ABB RobotStudio station: TFM_Robot.rspag

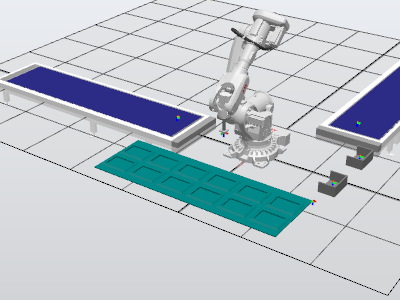
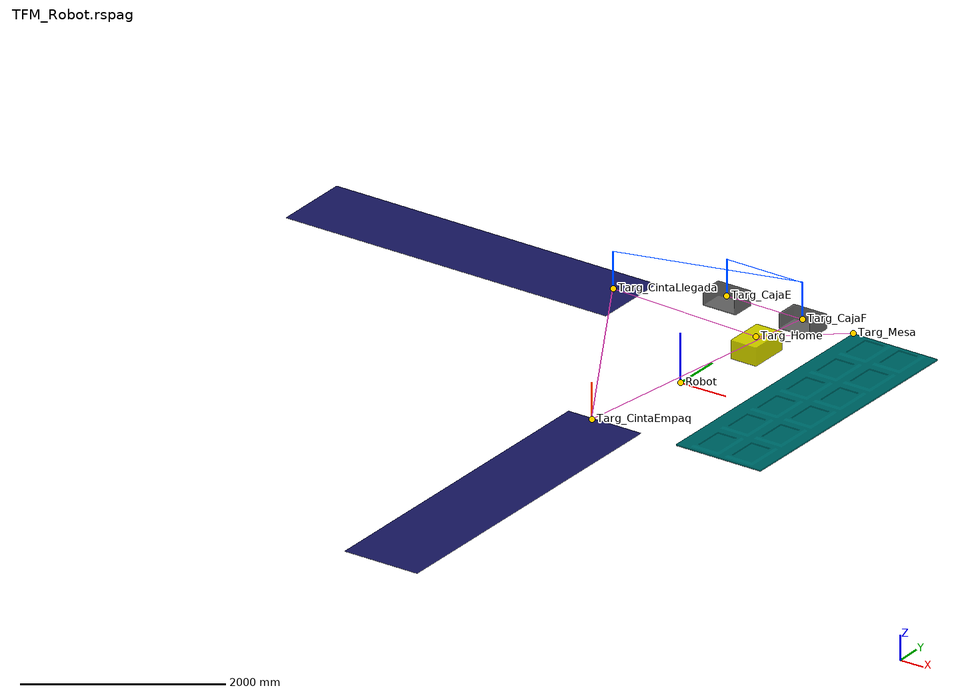
[picture v1: parts stored in the station drawn from their meshes, with robot base, taught points and paths (robot models come from the ABB library and are not in the file)]
--- station ---
Station TFM_Robot (saved by RobotStudio 24.2.10789.0)
Controller Controller_TFM
  mechanical unit ROB_1: Robot, 6 joints, base frame (0, 0, 0) mm
Layout (positions relative to the parent item):
  - Robot [mechanism] at (0, 0, 0) mm; joint values [0, -0.3937, 1.1224, 0, 0.8422, 1.5708] (rad or m)
      links: Base, Link1, Link2, Link3, Link4, Link5, Link6, LinkD1, LinkD2
  - GarraVentosas [mechanism] at (900, 0, 990) mm, rotated rx -180 ry 0 rz 90 deg
      TCP GarraVentosas at (0, 0, 240) mm
      links: GarraVentosas
  - MesaTrabajo [part] at (2000, 1500, 200) mm, rotated rx 90 ry 0 rz -90 deg, size 3000 x 35 x 1000 mm
  - CintaEmpaquetadora [part, from %ABB.RobotStudio.Models.Conveyors%\Conveyor 950 4000 h2.rslib] at (-455, -1200.38, -340.52) mm, rotated rx 0 ry 0 rz -90 deg
  - sup_CintaEmp [part] at (440.42, -1293.73, 94.49) mm, rotated rx 0 ry 0 rz 180 deg, size 864.5 x 3800 x 0 mm
  - sup_CintaGeneral [part] at (-1308.17, 600.35, 117.18) mm, rotated rx 0 ry 0 rz 90 deg, size 864.5 x 3800 x 0 mm
  - CintaGeneral [part, from %ABB.RobotStudio.Models.Conveyors%\Conveyor 950 4000 h2.rslib] at (-1231.46, 1484.09, -320.73) mm, rotated rx 0 ry 0 rz 180 deg
  - Surtidores_Cajas [part] at (205, 1630, 100) mm, rotated rx 90 ry 0 rz 0 deg, size 390 x 160 x 260 mm
  - Surtidores [part] at (-695, 1630, 100) mm, rotated rx 90 ry 0 rz 0 deg, size 390 x 160 x 260 mm
  - Ventosas [smart component] at (900, 0, 750) mm, rotated rx -180 ry 0 rz 90 deg
      signals: DI DI_Vacio, DI DI_Soplar, DO DO_Pieza, DI DI_VacioCaja, DI DI_SoplarCajas
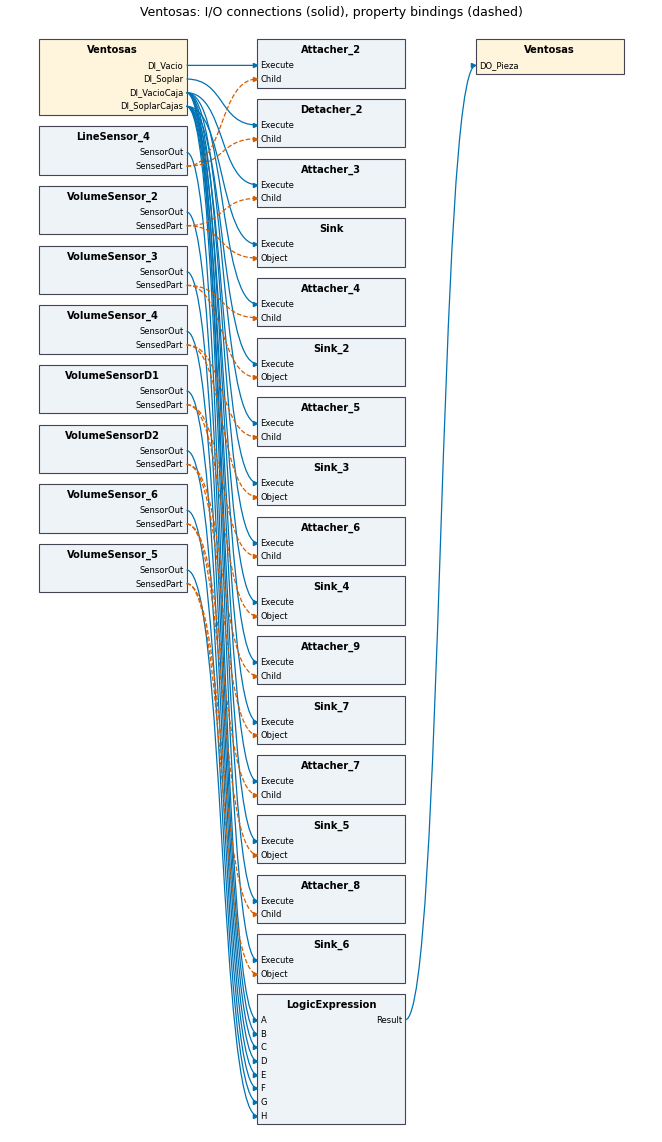
      connections:
        Ventosas.DI_Vacio -> Attacher_2.Execute
        Ventosas.DI_Soplar -> Detacher_2.Execute
        Ventosas.DI_VacioCaja -> Attacher_3.Execute
        Ventosas.DI_VacioCaja -> Attacher_4.Execute
        Ventosas.DI_VacioCaja -> Attacher_5.Execute
        Ventosas.DI_VacioCaja -> Attacher_6.Execute
        Ventosas.DI_VacioCaja -> Attacher_7.Execute
        Ventosas.DI_VacioCaja -> Attacher_8.Execute
        Ventosas.DI_SoplarCajas -> Sink.Execute
        Ventosas.DI_SoplarCajas -> Sink_2.Execute
        Ventosas.DI_SoplarCajas -> Sink_3.Execute
        Ventosas.DI_SoplarCajas -> Sink_4.Execute
        Ventosas.DI_SoplarCajas -> Sink_5.Execute
        Ventosas.DI_SoplarCajas -> Sink_6.Execute
        Ventosas.DI_VacioCaja -> Attacher_9.Execute
        Ventosas.DI_SoplarCajas -> Sink_7.Execute
        LineSensor_4.SensorOut -> LogicExpression.A
        VolumeSensor_2.SensorOut -> LogicExpression.B
        VolumeSensor_3.SensorOut -> LogicExpression.C
        VolumeSensor_4.SensorOut -> LogicExpression.D
        VolumeSensorD1.SensorOut -> LogicExpression.E
        VolumeSensorD2.SensorOut -> LogicExpression.F
        VolumeSensor_6.SensorOut -> LogicExpression.G
        VolumeSensor_5.SensorOut -> LogicExpression.H
        LogicExpression.Result -> Ventosas.DO_Pieza
        LineSensor_4.SensedPart => Attacher_2.Child
        LineSensor_4.SensedPart => Detacher_2.Child
        VolumeSensor_2.SensedPart => Attacher_3.Child
        VolumeSensor_2.SensedPart => Sink.Object
        VolumeSensor_3.SensedPart => Attacher_4.Child
        VolumeSensor_3.SensedPart => Sink_2.Object
        VolumeSensor_4.SensedPart => Attacher_5.Child
        VolumeSensor_4.SensedPart => Sink_3.Object
        VolumeSensorD1.SensedPart => Attacher_6.Child
        VolumeSensor_6.SensedPart => Attacher_7.Child
        VolumeSensor_5.SensedPart => Attacher_8.Child
        VolumeSensor_5.SensedPart => Sink_6.Object
        VolumeSensor_6.SensedPart => Sink_5.Object
        VolumeSensorD1.SensedPart => Sink_4.Object
        VolumeSensorD2.SensedPart => Attacher_9.Child
        VolumeSensorD2.SensedPart => Sink_7.Object
    - LineSensor_4 [smart component, from Components\LineSensor.rslib]
        properties: Start=[0.0199999999999999 0.02 -0.00999999999999998]; End=[0.0199999999999999 0.02 0.1]; Length=0.11; Radius=0.00476190476190476; Tag=(none); SensedPart=(none); SensedPoint=[0 0 0]
      - _sensorPart_ [part], size 9.5 x 9.5 x 110 mm
    - Attacher_2 [smart component, from Components\Attacher.rslib]
        properties: Parent=GarraVentosas; Flange=0; Child=(none); Mount=false; Offset=[0 0 0]; Orientation=[0 0 0]
    - Detacher_2 [smart component, from Components\Detacher.rslib]
        properties: Child=(none); KeepPosition=true
    - VolumeSensor_2 [smart component, from Components\VolumeSensor.rslib]
        properties: CornerPoint=[-0.220000006556705 -0.15000001063277 -0.00999992197537303]; Orientation=[0 0 0]; Length=0.44; Width=0.3; Height=0.2; Tag=PiezaA; PartialHit=true; SensedPart=(none)
      - _sensorPart_ [part], size 440 x 300 x 200 mm
    - VolumeSensor_3 [smart component, from Components\VolumeSensor.rslib] at (-100, 0, 0) mm
        properties: CornerPoint=[-0.120000006556705 -0.150000009019282 -0.00999992620903045]; Orientation=[0 0 0]; Length=0.44; Width=0.3; Height=0.2; Tag=PiezaB; PartialHit=true; SensedPart=(none)
      - _sensorPart_ [part], size 440 x 300 x 200 mm
    - VolumeSensor_4 [smart component, from Components\VolumeSensor.rslib] at (-200, 0, 0) mm
        properties: CornerPoint=[-0.0200000065567047 -0.150000007405794 -0.00999993044268799]; Orientation=[0 0 0]; Length=0.44; Width=0.3; Height=0.2; Tag=PiezaC; PartialHit=true; SensedPart=(none)
      - _sensorPart_ [part], size 440 x 300 x 200 mm
    - VolumeSensor_5 [smart component, from Components\VolumeSensor.rslib] at (-300, 0, 0) mm
        properties: CornerPoint=[0.0799999934432951 -0.150000005792307 -0.00999993467634541]; Orientation=[0 0 0]; Length=0.44; Width=0.3; Height=0.2; Tag=PiezaF; PartialHit=true; SensedPart=(none)
      - _sensorPart_ [part], size 440 x 300 x 200 mm
    - VolumeSensor_6 [smart component, from Components\VolumeSensor.rslib] at (-400, 0, 0) mm
        properties: CornerPoint=[0.179999993443295 -0.150000004178819 -0.00999993891000295]; Orientation=[0 0 0]; Length=0.44; Width=0.3; Height=0.2; Tag=PiezaE; PartialHit=true; SensedPart=(none)
      - _sensorPart_ [part], size 440 x 300 x 200 mm
    - VolumeSensorD1 [smart component, from Components\VolumeSensor.rslib] at (-500, 0, 0) mm
        properties: CornerPoint=[0.279999993443295 -0.150000002565331 -0.00999994314366048]; Orientation=[0 0 0]; Length=0.44; Width=0.12; Height=0.2; Tag=PiezaD; PartialHit=true; SensedPart=(none)
      - _sensorPart_ [part], size 440 x 120 x 200 mm
    - Attacher_3 [smart component, from Components\Attacher.rslib]
        properties: Parent=GarraVentosas; Flange=0; Child=(none); Mount=false; Offset=[0 0 0]; Orientation=[0 0 0]
    - Attacher_4 [smart component, from Components\Attacher.rslib]
        properties: Parent=GarraVentosas; Flange=0; Child=(none); Mount=false; Offset=[0 0 0]; Orientation=[0 0 0]
    - Attacher_5 [smart component, from Components\Attacher.rslib]
        properties: Parent=GarraVentosas; Flange=0; Child=(none); Mount=false; Offset=[0 0 0]; Orientation=[0 0 0]
    - Sink [smart component, from Components\Sink.rslib]
        properties: Object=(none)
    - Sink_2 [smart component, from Components\Sink.rslib]
        properties: Object=(none)
    - Sink_3 [smart component, from Components\Sink.rslib]
        properties: Object=(none)
    - Attacher_6 [smart component, from Components\Attacher.rslib]
        properties: Parent=GarraVentosas; Flange=0; Child=(none); Mount=false; Offset=[0 0 0]; Orientation=[0 0 0]
    - Attacher_7 [smart component, from Components\Attacher.rslib]
        properties: Parent=GarraVentosas; Flange=0; Child=(none); Mount=false; Offset=[0 0 0]; Orientation=[0 0 0]
    - Attacher_8 [smart component, from Components\Attacher.rslib]
        properties: Parent=GarraVentosas; Flange=0; Child=(none); Mount=false; Offset=[0 0 0]; Orientation=[0 0 0]
    - Sink_4 [smart component, from Components\Sink.rslib]
        properties: Object=(none)
    - Sink_5 [smart component, from Components\Sink.rslib]
        properties: Object=(none)
    - Sink_6 [smart component, from Components\Sink.rslib]
        properties: Object=(none)
    - VolumeSensorD2 [smart component, from Components\VolumeSensor.rslib] at (-400, 0, 0) mm
        properties: CornerPoint=[0.180000001768298 0.0299999953642274 -0.00999992383046211]; Orientation=[-1.22460538918519E-16 -4.56955773775466E-08 -4.37113878525484E-08]; Length=0.44; Width=0.12; Height=0.2; Tag=PiezaD; PartialHit=true; SensedPart=(none)
      - _sensorPart_ [part], size 440 x 120 x 200 mm
    - Attacher_9 [smart component, from Components\Attacher.rslib]
        properties: Parent=GarraVentosas; Flange=0; Child=(none); Mount=false; Offset=[0 0 0]; Orientation=[0 0 0]
    - Sink_7 [smart component, from Components\Sink.rslib]
        properties: Object=(none)
    - LogicExpression [smart component, from Components\LogicExpression.rslib]
        properties: Expression=A OR B OR C OR D OR E OR F OR G OR H
  - ReponedorPiezas [smart component]
      signals: DI DI_Pieza0, DI DI_Pieza1, DI DI_Pieza2, DI DI_Pieza3, DI DI_Pieza4, DI DI_Pieza5
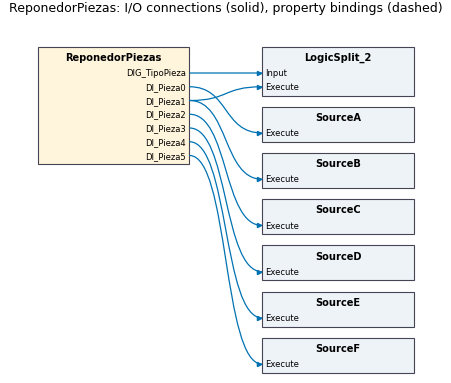
      connections:
        ReponedorPiezas.DIG_TipoPieza -> LogicSplit_2.Input
        ReponedorPiezas.DI_Pieza0 -> SourceA.Execute
        ReponedorPiezas.DI_Pieza1 -> Source_2.Execute
        ReponedorPiezas.DI_Pieza1 -> SourceB.Execute
        ReponedorPiezas.DI_Pieza2 -> SourceC.Execute
        ReponedorPiezas.DI_Pieza3 -> SourceD.Execute
        ReponedorPiezas.DI_Pieza4 -> SourceE.Execute
        ReponedorPiezas.DI_Pieza5 -> SourceF.Execute
    - SourceA [smart component, from Components\Source.rslib]
        properties: Source=PiezaA; Copy=(none); Parent=(none); Position=[-1.499 0.993 0.16]; Orientation=[0 0 -1.5707963267949]; Transient=true; PhysicsBehavior=-1
    - SourceB [smart component, from Components\Source.rslib]
        properties: Source=PiezaB; Copy=(none); Parent=(none); Position=[-1.5 1 0.16]; Orientation=[0 0 -1.5707963267949]; Transient=true; PhysicsBehavior=-1
    - SourceC [smart component, from Components\Source.rslib]
        properties: Source=PiezaC; Copy=(none); Parent=(none); Position=[-1.5 1 0.16]; Orientation=[0 0 -1.5707963267949]; Transient=true; PhysicsBehavior=-1
    - SourceD [smart component, from Components\Source.rslib]
        properties: Source=PiezaD; Copy=(none); Parent=(none); Position=[-1.5 1 0.16]; Orientation=[0 0 -1.5707963267949]; Transient=true; PhysicsBehavior=-1
    - SourceE [smart component, from Components\Source.rslib]
        properties: Source=PiezaE; Copy=(none); Parent=(none); Position=[-0.5015 1.502 0.176751]; Orientation=[0 0 -1.5707963267949]; Transient=true; PhysicsBehavior=-1
    - SourceF [smart component, from Components\Source.rslib]
        properties: Source=PiezaF; Copy=(none); Parent=(none); Position=[0.3995 1.501 0.18]; Orientation=[0 0 -1.5707963267949]; Transient=true; PhysicsBehavior=-1
    - PiezaA [part] at (-1500, 1000, 160) mm, size 130 x 210 x 80 mm
    - PiezaB [part] at (-1500, 1000, 160) mm, size 96.5 x 100 x 80 mm
    - PiezaC [part] at (-1500, 1000, 160) mm, size 96.5 x 100 x 80 mm
    - PiezaD [part] at (-1500, 1000, 160) mm, size 100 x 100 x 80 mm
    - PiezaE [part] at (-500, 1500, 176.75) mm, rotated rx 0 ry 0 rz -90 deg, size 230 x 340 x 34 mm
    - PiezaF [part] at (400, 1500, 180) mm, rotated rx 0 ry 0 rz -90 deg, size 230 x 340 x 58 mm
Attachment: sup_CintaGeneral is attached to CintaGeneral
Attachment: sup_CintaEmp is attached to CintaEmpaquetadora
Attachment: Ventosas is attached to GarraVentosas / GarraVentosas
Attachment: GarraVentosas is attached to Robot / Link6
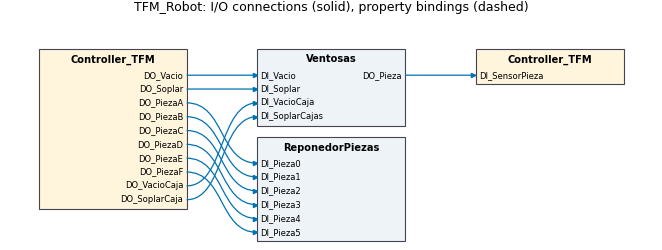
Station logic (signal -> signal, property => property):
  Ventosas.DO_Pieza -> Controller_TFM.DI_SensorPieza
  Controller_TFM.DO_Vacio -> Ventosas.DI_Vacio
  Controller_TFM.DO_Soplar -> Ventosas.DI_Soplar
  Controller_TFM.DO_PiezaA -> ReponedorPiezas.DI_Pieza0
  Controller_TFM.DO_PiezaB -> ReponedorPiezas.DI_Pieza1
  Controller_TFM.DO_PiezaC -> ReponedorPiezas.DI_Pieza2
  Controller_TFM.DO_PiezaD -> ReponedorPiezas.DI_Pieza3
  Controller_TFM.DO_PiezaE -> ReponedorPiezas.DI_Pieza4
  Controller_TFM.DO_PiezaF -> ReponedorPiezas.DI_Pieza5
  Controller_TFM.DO_VacioCaja -> Ventosas.DI_VacioCaja
  Controller_TFM.DO_SoplarCaja -> Ventosas.DI_SoplarCajas
Targets, tools, work objects and paths stored in the station and not in the controller backup, written as RAPID:
! task T_ROB1
MODULE Module1
  PROC processTCP()
    ErrorRX;
    ErrorRX;
    PulseDO \High\PLength:=0.5,DO_PiezaA;
    PulseDO \High\PLength:=0.5,DO_PiezaB;
    PulseDO \High\PLength:=0.5,DO_PiezaC;
    PulseDO \High\PLength:=0.5,DO_PiezaD;
    PulseDO \High\PLength:=0.5,DO_PiezaD;
    PulseDO \High\PLength:=0.5,DO_PiezaE;
    PulseDO \High\PLength:=0.5,DO_PiezaF;
    ErrorRX;
    ErrorRX;
    ErrorRX;
    ErrorRX;
    ErrorRX;
  ENDPROC
  PROC ErrorRX()
    PulseDO \High\PLength:=1,DO_ErrorRX;
  ENDPROC
ENDMODULE


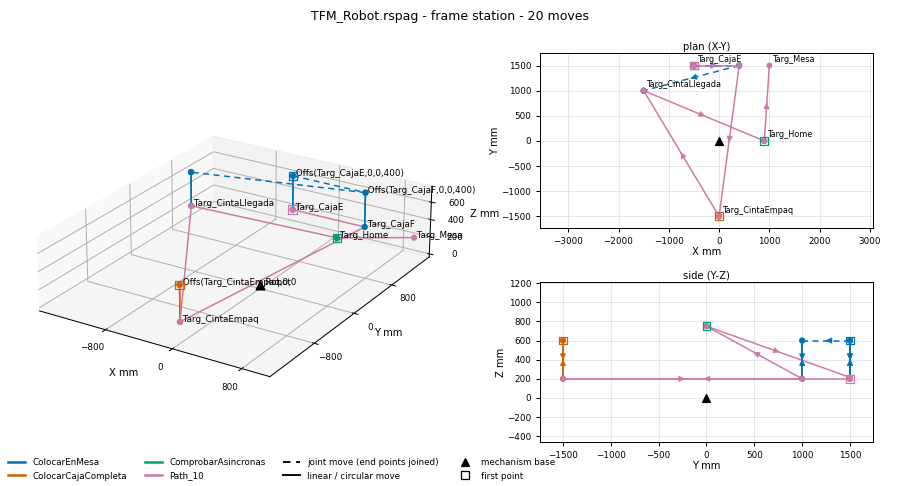
[picture p0: tool path of TFM_Robot.rspag in frame station, 20 of 26 moves have a stored position in this frame; points joined in program order, loops and branches not executed]
--- Backups/Controller_TFM/RAPID/TASK1/PROGMOD/CalibData.mod ---
MODULE CalibData
    PERS tooldata GarraVentosas:=[TRUE,[[0,0,240],[1,0,0,0]],[1,[0,0,1],[1,0,0,0],0,0,0]];
ENDMODULE

--- Backups/Controller_TFM/RAPID/TASK1/PROGMOD/Module1.mod ---
MODULE Module1
! Declaracion de los targets.
CONST robtarget Targ_CajaE:=[[-500,1500,200],[0,0,1,0],[1,0,1,0],[9E+09,9E+09,9E+09,9E+09,9E+09,9E+09]];
CONST robtarget Targ_CajaF:=[[400,1500,200],[0,0,1,0],[0,0,0,0],[9E+09,9E+09,9E+09,9E+09,9E+09,9E+09]];
CONST robtarget Targ_CintaEmpaq:=[[-0.000065567,-1500.000031808,200.000065078],[0,0,1,-0.000000008],[-2,0,-2,0],[9E+09,9E+09,9E+09,9E+09,9E+09,9E+09]];
CONST robtarget Targ_CintaLlegada:=[[-1500.000032056,1000.000001355,200.000069515],[-0.000000007,0,1,0.000000004],[1,0,1,0],[9E+09,9E+09,9E+09,9E+09,9E+09,9E+09]];
CONST robtarget Targ_Mesa:=[[999.999977515,1500.00004795,215.000069515],[0.000000008,0.707106781,0.707106781,0.000000002],[0,-1,1,0],[9E+09,9E+09,9E+09,9E+09,9E+09,9E+09]];
CONST robtarget Targ_Home:=[[900,0,750],[0,0.707106781,0.707106781,0],[0,0,0,0],[9E+09,9E+09,9E+09,9E+09,9E+09,9E+09]];

! Numero maximo de posiciones dentro de la mesa.
CONST num maximoNumMesas := 12;
! Numero maximo de materiales para los que el robot ha sido programado.
CONST num maximoNumMateriales := 5;

VAR socketdev serverSocket;
VAR socketdev clientSocket;
VAR bool servidorConectado := FALSE;
VAR string inputData;

! Almacena el numero de componentes (sin contar base y tapa) que maneja el robot.
VAR num numeroMateriales := maximoNumMateriales;
! Almacena el numero maximo de mesas que esta manejando el sistema en ese momento.
VAR num numeroMesas := maximoNumMesas;
! TRUE si hay algun material pegado a las ventosas. Variable necesaria por si falla la ventosa.
VAR bool transportandoMaterial := FALSE;

! Interrupcion para gestionar la deteccion de piezas.
VAR intnum int_DISensorPieza;

!**************************************************************************************************
! main() es la funcion de comienzo del programa. Si termina, se vuelve a ejecutar desde el
! comienzo.
!**************************************************************************************************
PROC main()
    ! Enlazar interrupcion con su funcion de interrupcion.
    CONNECT int_DISensorPieza WITH IntSensorPiezas;
    ! Disparar interrupcion unicamente cuando falle el sensor de piezas (pase de uno a cero la
    ! entrada DI_SensorPieza).
    ISignalDI DI_SensorPieza, 0, int_DISensorPieza;

    ! Esperar conexion entrante del PLC
    ConectarTCP;
    ! Mientras este conectado, realizar las peticiones del PLC.
    WHILE servidorConectado DO
        ProcesarMensajesTCP;
    ENDWHILE
ENDPROC

!**************************************************************************************************
! IntSensorPiezas es la funcion que se ejecuta cuando el sensor da un fallo mientras se esta
! transportando material.
!**************************************************************************************************
TRAP IntSensorPiezas
    IF transportandoMaterial THEN
        EscribirTCP "1?ACT";
        StopMove;
    ENDIF
ENDTRAP

!**************************************************************************************************
! ProcesarMensajesTCP() recibe los mensajes por TCP y realiza los movimientos u operaciones que
! el PLC instruya al robot.
!**************************************************************************************************
PROC ProcesarMensajesTCP()
    VAR bool msgOK;
    VAR num inputID;
    VAR num matDestino;
    VAR num mesaDestino;
    VAR bool mensajeRecibido;

    ! Recepcion de datos desde el TCP (bloquea el programa durante 10 segundos). Si no se recibe
    ! nada envia un mensaje para tratar de conectarse.
    mensajeRecibido := LeerTCP(10);
    IF NOT mensajeRecibido THEN
        ! Trata de reconectar.
        SolicitarConfiguracion;
        RETURN;
    ENDIF

    ! Convertir el numero inicial del mensaje a numero.
    msgOK := StrToVal(StrPart(inputData,1,1), inputID);
    IF NOT msgOK THEN
        ! Mandar mensaje de error de transmision.
        ErrorRX "ID";
        RETURN;
    ENDIF

    ! Coger material.
    IF inputID = 3 THEN
        IF StrLen(inputData) < 8 THEN
            ErrorRX "LEN";
            RETURN;
        ENDIF

        ! Obtener la ID del material que se desea coger.
        matDestino := ConvertirStringMaterial(StrPart(inputData,2,4));
        IF matDestino < 0  OR matDestino >= (numeroMateriales+2) THEN
            ! Error al parsear la ID del material.
            ErrorRX "MAT";
            RETURN;
        ENDIF

        ! Activar senales digitales para que ReponedorPiezas genere las piezas
        ! correspondientes.
        IF matDestino = numeroMateriales THEN
            PulseDO \High,\PLength:=0.5, DO_PiezaE;
        ELSEIF matDestino = numeroMateriales+1 THEN
            PulseDO \High,\PLength:=0.5, DO_PiezaF;
        ELSEIF matDestino = 0 THEN
            PulseDO \High,\PLength:=0.5, DO_PiezaA;
        ELSEIF matDestino = 1 THEN
            PulseDO \High,\PLength:=0.5, DO_PiezaB;
        ELSEIF matDestino = 2 THEN
            PulseDO \High,\PLength:=0.5, DO_PiezaC;
        ELSEIF matDestino = 3 THEN
            PulseDO \High,\PLength:=0.5, DO_PiezaD;
        ELSEIF matDestino = 4 THEN
            PulseDO \High,\PLength:=0.5, DO_PiezaD;
        ELSE
            ! Mandar mensaje de error fatal, no deberia ser posible entrar aqui.
            ErrorRX "FATAL";
            RETURN;
        ENDIF

        ! Obtener la ID de la mesa destino de la pieza.
        mesaDestino := StrToByte(StrPart(inputData,7,2)\Hex);
        IF mesaDestino >= maximoNumMesas THEN
            ErrorRX "MESA";
            RETURN;
        ENDIF

        ! Enviar el ACK.
        EscribirTCP "0ACK3";

        ! Comprobacion rapida por si hay un mensaje para detener el programa.
        mensajeRecibido := LeerTCP(0.5);
        IF mensajeRecibido THEN
            ! Convertir el numero inicial del mensaje a numero.
            msgOK := StrToVal(StrPart(inputData,1,1), inputID);
            IF NOT msgOK THEN
                ! Mandar mensaje de error de transmision.
                ErrorRX "ID";
                RETURN;
            ENDIF
            ComprobarAsincronas(inputID);
        ENDIF

        ! Algoritmo de posicionamiento de objetos en mesas.
        ColocarEnMesa matDestino, mesaDestino;

        ! Una vez colocado el objeto, manda senal de MaterialColocado.
        EscribirTCP "3MAT_COL";

    ! Coloca una caja completa en la cinta de empaquetado.
    ELSEIF inputID = 4 THEN
        IF StrLen(inputData) < 4 THEN
            ErrorRX "LEN";
            RETURN;
        ENDIF

        ! Obtener la ID de la posicion donde se encuentra la caja que se desea colocar
        ! en la cinta general.
        mesaDestino := StrToByte(StrPart(inputData,3,2)\Hex);
        IF mesaDestino > maximoNumMesas THEN
            ErrorRX "MESA";
            RETURN;
        ENDIF

        ! Enviar el ACK.
        EscribirTCP "0ACK4";

        ! Comprobacion rapida por si hay un mensaje para detener el programa.
        mensajeRecibido := LeerTCP(0.5);
        IF mensajeRecibido THEN
            ! Convertir el numero inicial del mensaje a numero.
            msgOK := StrToVal(StrPart(inputData,1,1), inputID);
            IF NOT msgOK THEN
                ! Mandar mensaje de error de transmision.
                ErrorRX "ID";
                RETURN;
            ENDIF
            ComprobarAsincronas(inputID);
        ENDIF

        ! Algoritmo de posicionamiento de cajas completas en la cinta de empaquetado.
        ColocarCajaCompleta mesaDestino;

        ! Una vez colocada la caja, manda senal de MaterialColocado.
        EscribirTCP "3MAT_COL";

    ! Ir a HOME y otras senales.
    ELSE
        ComprobarAsincronas(inputID);
    ENDIF
ENDPROC

!**************************************************************************************************
! ColocarEnMesa(num mat, num mesa) recibe la ID del material y de la mesa donde se desea colocar
! dicho material y genera las instrucciones de movimiento del brazo del robot.
!**************************************************************************************************
PROC ColocarEnMesa(num mat, num mesa)
    VAR num x;
    VAR num y;
    VAR num xPos;
    VAR num yPos;
    VAR robtarget posicionFinal;

    ! Obtener la posicion X,Y dentro de la mesa. La esquina superior izquierda desde el punto
    ! de vista de la cinta de empaquetado es el 0,0. El numero de la mesa se puede recalcular
    ! como X*6+Y.
    x := mesa DIV 6;
    y := mesa MOD 6;

    ! Obtener las esquinas de la posicion de la mesa que se indica. A partir de estas se
    ! desplazaran las coordenadas donde se encuentran individualmente las piezas con respecto la
    ! bandeja.
    xPos := 200 + x*400;
    yPos := 80 + y*500;

    ! Punto final donde se colocara el componente. En esta linea es la posicion de la esquina
    ! superior izquierda de la mesa que se esta pasando a esta funcion en referencia al mundo.
    posicionFinal := Offs(Targ_Mesa, xPos, -yPos, 0);

    ! Dependiendo del material, la posicion donde se colocara variara. Esto ira en referencia
    ! a la posicion calculada anteriormente.
    IF mat = numeroMateriales THEN
        ! Base de la caja.
        posicionFinal := Offs(posicionFinal, 115,-170,40);
    ELSEIF mat = numeroMateriales+1 THEN
        ! Tapadera de la caja.
        posicionFinal := Offs(posicionFinal, 115,-170,93);
    ELSEIF mat = 0 THEN
        posicionFinal := Offs(posicionFinal, 75,-225,85);
    ELSEIF mat = 1 THEN
        posicionFinal := Offs(posicionFinal, 177,-283,85);
    ELSEIF mat = 2 THEN
        posicionFinal := Offs(posicionFinal, 177,-167,85);
    ELSEIF mat = 3 THEN
        posicionFinal := Offs(posicionFinal, 60,-60,85);
    ELSEIF mat = 4 THEN
        posicionFinal := Offs(posicionFinal, 170,-60,85);
    ENDIF

    ! Seleccion de la posicion donde se recogera el material.
    IF mat = numeroMateriales THEN
        ! Posicion de recogida de la caja.
        MoveJ Offs(Targ_CajaE,0,0,400),v5000,z20,GarraVentosas\WObj:=wobj0;
        MoveL Targ_CajaE,v500,fine,GarraVentosas\WObj:=wobj0;
        PulseDO \High,\PLength:=0.5, DO_Vacio;
        transportandoMaterial := TRUE;
        MoveL Offs(Targ_CajaE,0,0,400),v1000,z20,GarraVentosas\WObj:=wobj0;
    ELSEIF mat = numeroMateriales+1 THEN
        ! Posicion de recogida de la tapa.
        MoveJ Offs(Targ_CajaF,0,0,400),v5000,z20,GarraVentosas\WObj:=wobj0;
        MoveL Targ_CajaF,v500,fine,GarraVentosas\WObj:=wobj0;
        PulseDO \High,\PLength:=0.5, DO_Vacio;
        transportandoMaterial := TRUE;
        MoveL Offs(Targ_CajaF,0,0,400),v1000,z20,GarraVentosas\WObj:=wobj0;
    ELSE
        ! Componentes de la cinta general.
        MoveJ Offs(Targ_CintaLlegada,0,0,400),v5000,z20,GarraVentosas\WObj:=wobj0;
        MoveL Targ_CintaLlegada,v500,fine,GarraVentosas\WObj:=wobj0;
        PulseDO \High,\PLength:=0.5, DO_Vacio;
        transportandoMaterial := TRUE;
        MoveL Offs(Targ_CintaLlegada,0,0,400),v1000,z20,GarraVentosas\WObj:=wobj0;
    ENDIF

    ! Mandar senal de material recogido.
    EscribirTCP "2MAT_REC";

    ! Dejar el material en la posicion final.
    MoveJ Offs(posicionFinal,0,0,400),v5000,z20,GarraVentosas\WObj:=wobj0;
    MoveL posicionFinal,v500,fine,GarraVentosas\WObj:=wobj0;
    PulseDO \High,\PLength:=0.5, DO_Soplar;
    transportandoMaterial := FALSE;
    MoveL Offs(posicionFinal,0,0,400),v1000,fine,GarraVentosas\WObj:=wobj0;
ENDPROC

!**************************************************************************************************
! ColocarCajaCompleta(num mat) coloca una caja completa en la cinta de empaquetado.
!**************************************************************************************************
PROC ColocarCajaCompleta(num mesa)
    VAR num x;
    VAR num y;
    VAR num xPos;
    VAR num yPos;
    VAR robtarget posicionFinal;

    ! Obtener la posicion X,Y dentro de la mesa. La esquina superior izquierda desde el punto
    ! de vista de la cinta de empaquetado es el 0,0. El numero de la mesa se puede recalcular
    ! como X*6+Y.
    x := mesa DIV 6;
    y := mesa MOD 6;

    ! Anadir la posicion del centro de la caja (115, 170); es decir, la mitad de las
    ! dimensiones.
    xPos := 200 + x*400 + 115;
    yPos := 80 + y*500 + 170;

    ! Posicion del centro de la caja en la mesa.
    posicionFinal := Offs(Targ_Mesa, xPos, -yPos, 93);

    MoveJ Offs(posicionFinal,0,0,400),v5000,z20,GarraVentosas\WObj:=wobj0;
    MoveL posicionFinal,v500,fine,GarraVentosas\WObj:=wobj0;
    PulseDO \High,\PLength:=0.5, DO_VacioCaja;
    transportandoMaterial := TRUE;
    MoveL Offs(posicionFinal,0,0,400),v1000,z20,GarraVentosas\WObj:=wobj0;

    ! Dejar el material en la cinta de empaquetado.
    MoveJ Offs(Targ_CintaEmpaq,0,0,400),v5000,z20,GarraVentosas\WObj:=wobj0;
    MoveL Targ_CintaEmpaq,v500,fine,GarraVentosas\WObj:=wobj0;
    transportandoMaterial := FALSE;
    PulseDO \High,\PLength:=0.5, DO_SoplarCaja;
    MoveL Offs(Targ_CintaEmpaq,0,0,400),v1000,fine,GarraVentosas\WObj:=wobj0;
ENDPROC

!**************************************************************************************************
! ConectarTCP() esta funcion realiza la conexion mediante TCP al socket del cliente. Una vez
! realizada la conexion, manda un mensaje con su configuracion inicial al PLC y espera una
! respuesta para confirmar que esta correctamente conectado.
!**************************************************************************************************
PROC ConectarTCP()
    ! Inicializacion de los sockets.
    SocketCreate serverSocket;
    SocketBind serverSocket, "127.0.0.1", 9876;
    SocketListen serverSocket;
    SocketAccept serverSocket, clientSocket,\Time:=WAIT_MAX;
    SolicitarConfiguracion;
ENDPROC

!**************************************************************************************************
! SolicitarConfiguracion() manda al PLC un mensaje con la configuracion actual del robot. Espera
! que el PLC le devuelva la configuracion que esta utilizando y la adopta si es valida.
!**************************************************************************************************
PROC SolicitarConfiguracion()
    VAR bool msgOK;
    VAR num inputID;

SolicitarConfig:
    ! Mandar mensaje de conexion completada junto con el numero m?ximo de mesas y materiales
    ! permitidos.
    EscribirTCP "405M0C";
    ! Espera la respuesta del sistema con la configuracion.
    msgOK := LeerTCP(5);
    IF NOT msgOK THEN
        GOTO SolicitarConfig;
    ENDIF

    ! Comprobar la longitud de la cadena.
    IF StrLen(inputData) < 6 THEN
        ErrorRX("LEN");
        GOTO SolicitarConfig;
    ENDIF

    ! Comprobar que la ID es la de Parametros.
    msgOK := StrToVal(StrPart(inputData,1,1), inputID);
    IF inputID <> 5 THEN
        GOTO SolicitarConfig;
    ENDIF

    ! Obtener el numero maximo de materiales por bandeja.
    numeroMateriales := StrToByte(StrPart(inputData,2,2)\Hex);
    IF numeroMateriales > maximoNumMateriales THEN
        ErrorRX("CONF_MAT");
        GOTO SolicitarConfig;
    ENDIF

    ! Obtener el numero de mesas que puede haber.
    numeroMesas := StrToByte(StrPart(inputData,5,2)\Hex);
    IF numeroMesas > maximoNumMesas THEN
        ErrorRX("CONF_MESA");
        GOTO SolicitarConfig;
    ENDIF

    ! Enviar ACK. La conexion con el PLC ya ha sido establecida.
    EscribirTCP "0ACK5";
    servidorConectado := TRUE;
ENDPROC

!**************************************************************************************************
! ErrorRX(string errMsg) es una funcion que envia al PLC un mensaje de error tras la recepcion de
! un mensaje que el PLC ha mandado.
!**************************************************************************************************
PROC ErrorRX(string errMsg)
    EscribirTCP "1?"+errMsg;
    PulseDO \High,\PLength:=1, DO_ErrorRX;
ENDPROC

!**************************************************************************************************
! Reconectar() cierra los sockets y vuelve a intentar realizar una conexion con el PLC.
!**************************************************************************************************
PROC Reconectar()
    SocketClose serverSocket;
    SocketClose clientSocket;
    servidorConectado := FALSE;
    ConectarTCP;
ENDPROC

!**************************************************************************************************
! bool LeerTCP(num time) sirve para recibir un mensaje del PLC mediante TCP. Puede ser especificado
! un tiempo limite de espera, tras el cual se lanza una excepcion que es recogida en la seccion de
! ERROR. Devuelve true cuando el mensaje recibido es valido y false si no se ha recibido ningun
! mensaje antes de que acabe el tiempo de espera. Si el socket se desconecta intenta reconectarse
! y vuelve a leer el TCP.
!**************************************************************************************************
FUNC bool LeerTCP(num time)
    ! Comprobacion rapida por si hay un mensaje para detener el programa.
    SocketReceive clientSocket, \Str:=inputData, \Time:=time;
    RETURN TRUE;
ERROR
    IF ERRNO=ERR_SOCK_TIMEOUT THEN
        RETURN FALSE;
    ELSEIF ERRNO=ERR_SOCK_CLOSED THEN
        Reconectar;
        RETRY;
    ELSE
        ! Error desconocido, el sistema se apagara.
        Stop;
    ENDIF
ENDFUNC

!**************************************************************************************************
! EscribirTCP(string data) escribe por TCP mensajes hacia el PC. Si el socket se desconectara
! trata de reconectarse y vuelve a lanzar el mensaje.
!**************************************************************************************************
PROC EscribirTCP(string data)
    SocketSend clientSocket \Str:=data;
ERROR
    IF ERRNO=ERR_SOCK_CLOSED THEN
        Reconectar;
        RETRY;
    ELSE
        ! Error desconocido, el sistema se apagara.
        Stop;
    ENDIF
ENDPROC

!**************************************************************************************************
! ComprobarAsincronas(num inputID) procesa aquellos mensajes que no estan relacionados con el
! funcionamiento normal del sistema; por ejemplo, las instrucciones enviadas por operarios desde
! el HMI.
!**************************************************************************************************
PROC ComprobarAsincronas(num inputID)
    VAR bool msgOK;

    ! Estado del sistema. Mandar simplemente un ack.
    IF inputID = 2 THEN
        EscribirTCP "0ACK2";
    ! Parametros de configuracion.
    ELSEIF inputID = 5 THEN
        ! Comprobar la longitud de la cadena.
        IF StrLen(inputData) < 6 THEN
            ErrorRX("LEN");
            RETURN;
        ENDIF

        ! Comprobar que la ID es la de Parametros.
        msgOK := StrToVal(StrPart(inputData,1,1), inputID);
        IF inputID <> 5 THEN
            RETURN;
        ENDIF

        ! Comprobar que el numero de materiales por bandeja no supera el maximo.
        numeroMateriales := StrToByte(StrPart(inputData,2,2)\Hex);
        IF numeroMateriales > maximoNumMateriales THEN
            ErrorRX("NUM_MAT");
            RETURN;
        ENDIF

        ! Comprobar que el numero de mesas no supera el maximo.
        numeroMesas := StrToByte(StrPart(inputData,5,2)\Hex);
        IF numeroMesas > maximoNumMesas THEN
            ErrorRX("NUM_MES");
            RETURN;
        ENDIF

        EscribirTCP "0ACK5";
        servidorConectado := TRUE;

    ! Ir a HOME
    ELSEIF inputID = 6 THEN
        ! Enviar el ACK.
        EscribirTCP "0ACK6";

        MoveJ Targ_Home,v500,fine,GarraVentosas\WObj:=wobj0;

    ! Apagar la maquina
    ELSEIF inputID = 7 THEN
        ! Enviar el ACK.
        EscribirTCP "0ACK7";
        ! Ir a home y apagar.
        MoveJ Targ_Home,v500,fine,GarraVentosas\WObj:=wobj0;
        Stop;
    ENDIF
ENDPROC

!**************************************************************************************************
! num ConvertirStringMaterial(string strMat) recibe un string con el identificador del material y
! lo convierte a un numero que reconoce el robot. En caso de haber algun error, devuelve -1.
!**************************************************************************************************
FUNC num ConvertirStringMaterial(string strMat)
    VAR num numMatEntrada;
    VAR num numMat := 0;
    numMatEntrada := BitLsh(StrToByte(StrPart(strMat,1,2)\Hex),8) +
                     StrToByte(StrPart(strMat,3,2)\Hex);
    WHILE BitAnd(numMatEntrada, 1) = 0 DO
        numMatEntrada := BitRsh(numMatEntrada, 1);
        numMat := numMat + 1;
    ENDWHILE

    IF BitRsh(numMatEntrada, 1) <> 0 THEN
        RETURN -1;
    ENDIF
    RETURN numMat;
ENDFUNC

!**************************************************************************************************
! Funcion no utilizada. Sirve para poder transferir puntos desde la ventanda de posicion inicial
! a RAPID.
!**************************************************************************************************
PROC Path_10()
    MoveL Targ_CajaE,v500,z20,GarraVentosas\WObj:=wobj0;
    MoveL Targ_CajaF,v500,z20,GarraVentosas\WObj:=wobj0;
    MoveL Targ_CintaEmpaq,v500,z20,GarraVentosas\WObj:=wobj0;
    MoveL Targ_CintaLlegada,v500,z20,GarraVentosas\WObj:=wobj0;
    MoveL Targ_Home,v500,z20,GarraVentosas\WObj:=wobj0;
    MoveL Targ_Mesa,v500,z20,GarraVentosas\WObj:=wobj0;
ENDPROC

ENDMODULE

--- Backups/Controller_TFM/SYSPAR/EIO.cfg ---
EIO:CFG_1.0:6:1::
#
EIO_SIGNAL:

      -Name "DO_Vacio" -SignalType "DO" -Access "All"

      -Name "DO_Soplar" -SignalType "DO" -Access "All"

      -Name "DI_SensorPieza" -SignalType "DI" -Access "All"

      -Name "DO_PiezaA" -SignalType "DO" -Access "All"

      -Name "DO_PiezaB" -SignalType "DO" -Access "All"

      -Name "DO_PiezaC" -SignalType "DO" -Access "All"

      -Name "DO_PiezaD" -SignalType "DO" -Access "All"

      -Name "DO_PiezaE" -SignalType "DO" -Access "All"

      -Name "DO_PiezaF" -SignalType "DO" -Access "All"

      -Name "DO_ErrorRX" -SignalType "DO" -Access "All"

      -Name "DO_VacioCaja" -SignalType "DO" -Access "All"

      -Name "DO_SoplarCaja" -SignalType "DO" -Access "All"
